// TIA Portal V17 export
// export: Created 2025-06-26T06:49:27.1140034Z, ExportSetting WithDefaults, DisplayName Totally Integrated Automation Portal, DisplayVersion V17 Update 8, DisplayName TIA Portal Openness, DisplayVersion V17 Update 8, DisplayName TIA Portal Version Control Interface, DisplayVersion V17, DisplayName STEP 7 Professional, DisplayVersion V17 Update 8, DisplayName STEP 7 Safety, DisplayVersion V17 Update 6, DisplayName WinCC Advanced, DisplayVersion V17 Update 8
TYPE "CAN-IDs_ToSend"
// stored: IsFailsafeCompliant false
   STRUCT
      IDs : Array[0..74] of Int;
   END_STRUCT;
   // IDs[0] := 16#0201;
   // IDs[1] := 16#0202;
   // IDs[2] := 16#0203;
   // IDs[3] := 16#0204;
   // IDs[4] := 16#0205;
   // IDs[5] := 16#0206;
   // IDs[6] := 16#0207;
   // IDs[7] := 16#0210;
   // IDs[8] := 16#0220;
   // IDs[9] := 16#0221;
   // IDs[10] := 16#0222;
   // IDs[11] := 16#0223;
   // IDs[12] := 16#0224;
   // IDs[13] := 16#0240;
   // IDs[14] := 16#0241;
   // IDs[15] := 16#0242;
   // IDs[16] := 16#0243;
   // IDs[17] := 16#0501;
   // IDs[18] := 16#0244;
   // IDs[19] := 16#0245;
   // IDs[20] := 16#0246;
   // IDs[21] := 16#0250;
   // IDs[22] := 16#0251;
   // IDs[23] := 16#0252;
   // IDs[24] := 16#0253;
   // IDs[25] := 16#0254;
   // IDs[26] := 16#0260;
   // IDs[27] := 16#0261;
   // IDs[28] := 16#0262;
   // IDs[29] := 16#0263;
   // IDs[30] := 16#0264;
   // IDs[31] := 16#0301;
   // IDs[32] := 16#0302;
   // IDs[33] := 16#0310;
   // IDs[34] := 16#0311;
   // IDs[35] := 16#0312;
   // IDs[36] := 16#0313;
   // IDs[37] := 16#0314;
   // IDs[38] := 16#0320;
   // IDs[39] := 16#0321;
   // IDs[40] := 16#0322;
   // IDs[41] := 16#0323;
   // IDs[42] := 16#0324;
   // IDs[43] := 16#0241;
   // IDs[44] := 16#0243;
   // IDs[45] := 16#0501;
   // IDs[46] := 16#0401;
   // IDs[47] := 16#0402;
   // IDs[48] := 16#0403;
   // IDs[49] := 16#0404;
   // IDs[50] := 16#0405;
   // IDs[51] := 16#0451;
   // IDs[52] := 16#0452;
   // IDs[53] := 16#0453;
   // IDs[54] := 16#0454;
   // IDs[55] := 16#0455;
   // IDs[56] := 16#0456;
   // IDs[57] := 16#0457;
   // IDs[58] := 16#0458;
   // IDs[59] := 16#0459;
   // IDs[60] := 16#0460;
END_TYPE
